PROGRAM SevenSegmentDisplay
VAR
END_VAR

END_PROGRAM

(* stored: Version 1.1.0.1, ProductVersion 3.1.4024.12
   POU SevenSegmentDisplay: Id {8f9e204f-6405-4eea-b758-3a07a26e9b59}, SpecialFunc None *)
